ABB RobotStudio station: Project_2.rsstn

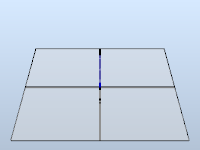
Station Station (saved by RobotStudio 21.1.9443.2)
Layout (positions relative to the parent item):
